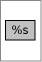
VISUALIZATION V_Rol  // 42x62
VAR_IN_OUT
	m_Input_fbRollo : FB_Rollo;
END_VAR
    Polygon (0,20)
    Polygon (0,20), invisible if: (m_Input_fbRollo.bOutRollo =0) <> 0
    Polygon (40,20), invisible if: (m_Input_fbRollo.bOutVisuAb =0) <> 0
    Polygon (40,40), invisible if: (m_Input_fbRollo.bOutVisuAb =1) <> 0
    Rectangle (5,20 30x20), "%s", text variable: m_Input_fbRollo.iActPos, colour toggle: (m_Input_fbRollo.bOutRollo) <> 0
    Polygon (40,20), colour toggle: (m_Input_fbRollo.bInVisuAuf) <> 0
        tap m_Input_fbRollo.bInVisuAuf
    Polygon (20,60), colour toggle: (m_Input_fbRollo.bInVisuAb) <> 0
        tap m_Input_fbRollo.bInVisuAb
END_VISUALIZATION

(* stored: Version 1.1.0.1, ProductVersion 3.1.4018.5
   Visu V_Rol: Id {63b97086-2633-450b-b944-f5a530c6e594} *)
